(* IEC 61131-3 sources: stc/pkg/parser/testdata, 8 files *)

(* ---- type_declarations.st ---- *)
TYPE MyEnum : (Red, Green := 1, Blue := 2); END_TYPE
TYPE MyStruct :
STRUCT
    x : INT;
    y : REAL;
    name : STRING(50);
END_STRUCT
END_TYPE
TYPE MyArray : ARRAY[1..10] OF INT; END_TYPE
TYPE MySubrange : INT(0..100); END_TYPE
TYPE MyAlias : DINT; END_TYPE

(* ---- error_recovery.st ---- *)
FUNCTION_BLOCK FB_Broken
VAR_INPUT
    x : BOOL;
END_VAR
IF x THEN
    y := ;
END_IF;
z := 42;
END_FUNCTION_BLOCK

(* ---- function_block_oop.st ---- *)
INTERFACE IMotor
METHOD Start : BOOL
END_METHOD
METHOD Stop : BOOL
END_METHOD
END_INTERFACE

FUNCTION_BLOCK FB_Motor EXTENDS FB_Base IMPLEMENTS IMotor
VAR
    _running : BOOL;
END_VAR
METHOD PUBLIC Start : BOOL
VAR_TEMP
    prev : BOOL;
END_VAR
    prev := _running;
    _running := TRUE;
    Start := NOT prev;
END_METHOD
METHOD PUBLIC OVERRIDE Stop : BOOL
    _running := FALSE;
    Stop := TRUE;
END_METHOD
PROPERTY Running : BOOL
END_PROPERTY
END_FUNCTION_BLOCK

(* ---- pointers_refs.st ---- *)
FUNCTION_BLOCK FB_PtrTest
VAR
    px : POINTER TO INT;
    rx : REFERENCE TO REAL;
    arr : ARRAY[0..9] OF POINTER TO BOOL;
END_VAR
    px^ := 42;
    rx := px^;
END_FUNCTION_BLOCK

(* ---- var_sections.st ---- *)
FUNCTION_BLOCK FB_VarTest
VAR_INPUT
    start : BOOL;
    speed : INT;
END_VAR
VAR_OUTPUT
    running : BOOL;
END_VAR
VAR_IN_OUT
    counter : INT;
END_VAR
VAR_TEMP
    temp : REAL;
END_VAR
VAR CONSTANT
    MAX_SPEED : INT := 100;
END_VAR
VAR RETAIN
    totalRuns : DINT;
END_VAR
END_FUNCTION_BLOCK

(* ---- control_flow.st ---- *)
PROGRAM ControlTest
VAR
    i : INT;
    x : INT;
    state : INT;
    flag : BOOL;
END_VAR
IF x > 10 THEN
    x := 0;
ELSIF x > 5 THEN
    x := x - 1;
ELSE
    x := x + 1;
END_IF;

CASE state OF
    0: x := 0;
    1..5: x := 1;
    10, 20, 30: x := 2;
ELSE
    x := -1;
END_CASE;

FOR i := 0 TO 10 BY 2 DO
    x := x + i;
END_FOR;

WHILE flag DO
    flag := FALSE;
END_WHILE;

REPEAT
    x := x + 1;
UNTIL x >= 100
END_REPEAT;
END_PROGRAM

(* ---- expressions.st ---- *)
PROGRAM ExprTest
VAR
    a, b, c, d : INT;
    f : BOOL;
END_VAR
    a := 1 + 2 * 3;
    b := (1 + 2) * 3;
    c := 2 ** 3 ** 2;
    d := a MOD b;
    f := a > 0 AND b < 100 OR c = d;
    f := NOT f XOR TRUE;
END_PROGRAM

(* ---- program_basic.st ---- *)
PROGRAM Main
VAR
    x : INT := 0;
    y : REAL := 3.14;
    name : STRING(80) := 'hello';
END_VAR
    x := x + 1;
    y := REAL#2.0 * y;
END_PROGRAM
